TYPE ST_Position :
STRUCT
	X	:	LREAL;
	Y	: 	LREAL;
	Z	: 	LREAL;
	C	: 	LREAL;
	A	: 	LREAL;
	rotX: 	LREAL;
	rotY: 	LREAL;
	rotZ: 	LREAL;
END_STRUCT
END_TYPE

(* stored: Version 1.1.0.1, ProductVersion 3.1.4024.3
   DUT ST_Position: Id {54512147-6c2e-4106-bc2c-b21f46de2f63} *)
